// Mitsubishi GX Works2 project: 梯形图   PLC: FX3U/FX3UC

PROGRAM MAIN
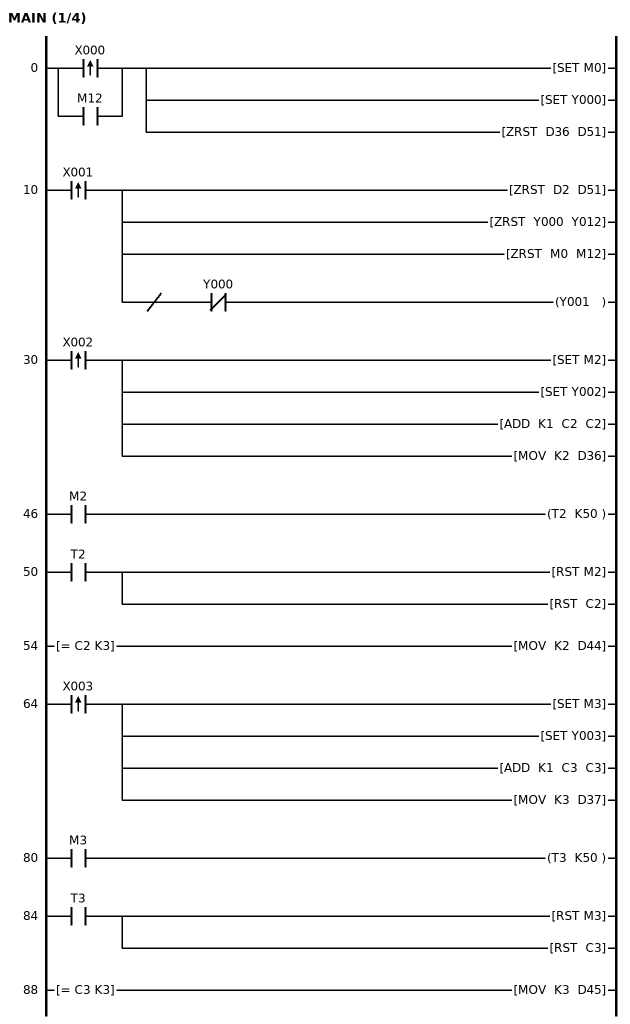
0     LDP     X000
      OR      M12
      SET     M0
      SET     Y000
      ZRST    D36 D51
10    LDP     X001
      ZRST    D2 D51
      ZRST    Y000 Y012
      ZRST    M0 M12
      INV
      ANI     Y000
      OUT     Y001
30    LDP     X002
      SET     M2
      SET     Y002
      ADD     K1 C2 C2
      MOV     K2 D36
46    LD      M2
      OUT     T2 K50
50    LD      T2
      RST     M2
      RST     C2
54    LD=     C2 K3
      MOV     K2 D44
64    LDP     X003
      SET     M3
      SET     Y003
      ADD     K1 C3 C3
      MOV     K3 D37
80    LD      M3
      OUT     T3 K50
84    LD      T3
      RST     M3
      RST     C3
88    LD=     C3 K3
      MOV     K3 D45
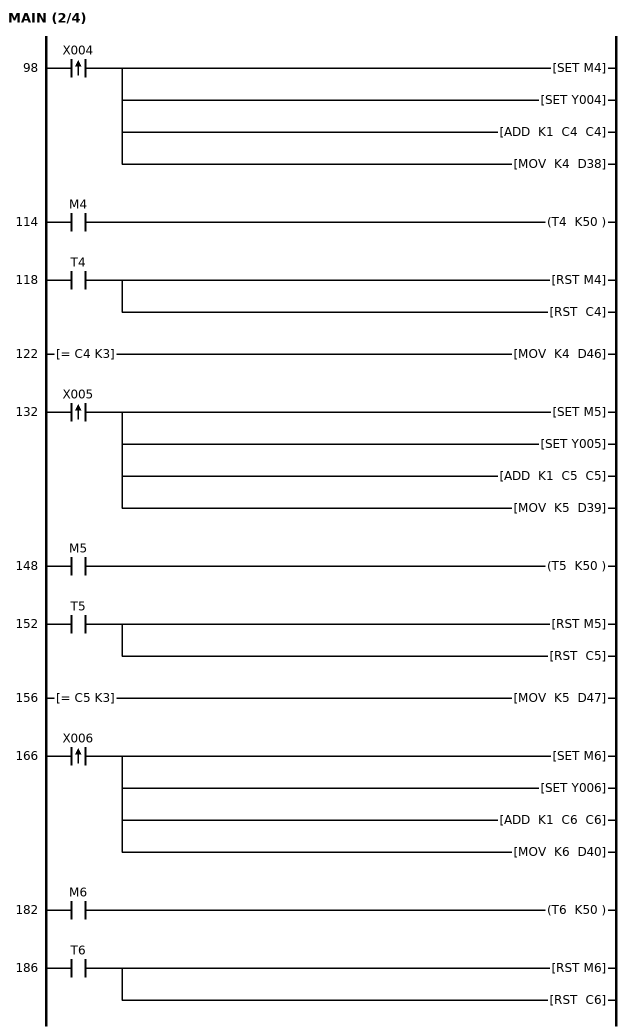
98    LDP     X004
      SET     M4
      SET     Y004
      ADD     K1 C4 C4
      MOV     K4 D38
114   LD      M4
      OUT     T4 K50
118   LD      T4
      RST     M4
      RST     C4
122   LD=     C4 K3
      MOV     K4 D46
132   LDP     X005
      SET     M5
      SET     Y005
      ADD     K1 C5 C5
      MOV     K5 D39
148   LD      M5
      OUT     T5 K50
152   LD      T5
      RST     M5
      RST     C5
156   LD=     C5 K3
      MOV     K5 D47
166   LDP     X006
      SET     M6
      SET     Y006
      ADD     K1 C6 C6
      MOV     K6 D40
182   LD      M6
      OUT     T6 K50
186   LD      T6
      RST     M6
      RST     C6
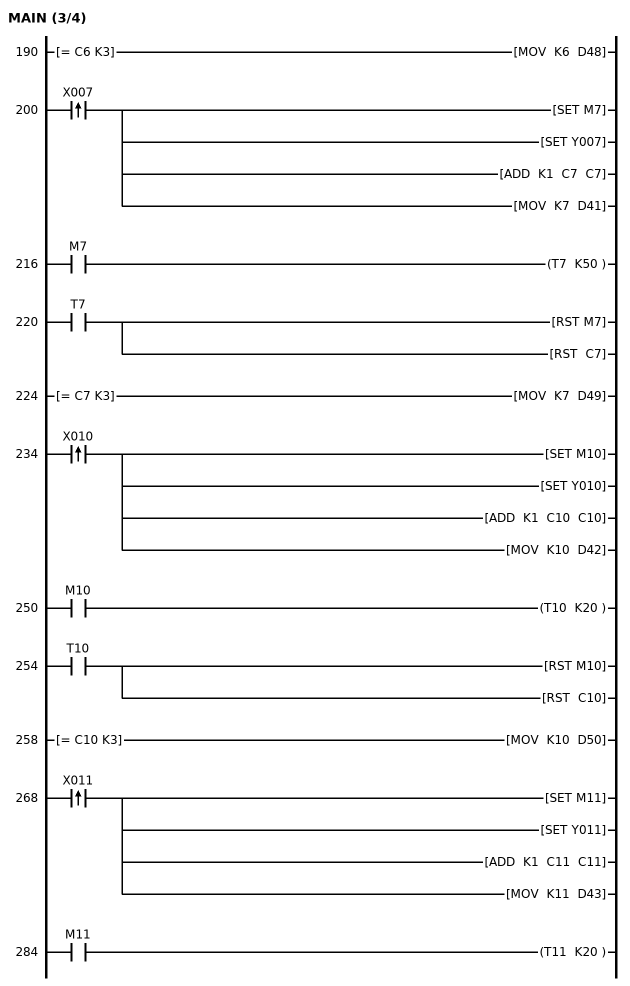
190   LD=     C6 K3
      MOV     K6 D48
200   LDP     X007
      SET     M7
      SET     Y007
      ADD     K1 C7 C7
      MOV     K7 D41
216   LD      M7
      OUT     T7 K50
220   LD      T7
      RST     M7
      RST     C7
224   LD=     C7 K3
      MOV     K7 D49
234   LDP     X010
      SET     M10
      SET     Y010
      ADD     K1 C10 C10
      MOV     K10 D42
250   LD      M10
      OUT     T10 K20
254   LD      T10
      RST     M10
      RST     C10
258   LD=     C10 K3
      MOV     K10 D50
268   LDP     X011
      SET     M11
      SET     Y011
      ADD     K1 C11 C11
      MOV     K11 D43
284   LD      M11
      OUT     T11 K20
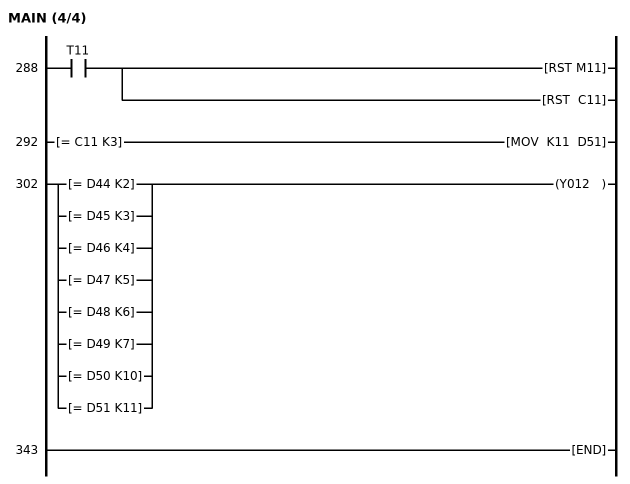
288   LD      T11
      RST     M11
      RST     C11
292   LD=     C11 K3
      MOV     K11 D51
302   LD=     D44 K2
      OR=     D45 K3
      OR=     D46 K4
      OR=     D47 K5
      OR=     D48 K6
      OR=     D49 K7
      OR=     D50 K10
      OR=     D51 K11
      OUT     Y012
343   END
END_PROGRAM
